FUNCTION_BLOCK FB113
TITLE = ''
AUTHOR : CB

VAR
	modes : FB41;
	fault : FB76;
	process : FB85;
	pilot : FB112;
END_VAR


BEGIN


NETWORK
TITLE =
//
//	modes
CALL #modes;



NETWORK
TITLE =
//
//	fault
CALL #fault;



NETWORK
TITLE =
//
//	process
CALL #process;



NETWORK
TITLE =
//
//	pilot
CALL #pilot;




END_FUNCTION_BLOCK
